TYPE ZComUnit :
STRUCT
{attribute '__ZwPlcApplicationComUnitDeclaration__'} // Do not remove this attribute! It is used for code generation.
END_STRUCT
END_TYPE

(* stored: Version 1.1.0.1
   DUT ZComUnit: Id {c82bcab2-9169-40c4-8c12-27bfd05a7c57} *)
